// TwinCAT 3 PLC project MotionTemplate
// ProgramVersion: 3.1.4024.0
// libraries:
//   Tc2_MC2, * (Beckhoff Automation GmbH)
//   Tc2_Standard, * (Beckhoff Automation GmbH)
//   Tc2_System, * (Beckhoff Automation GmbH)
//   Tc3_Module, * (Beckhoff Automation GmbH)
// project tree:
//   / PlcTask.TcTTO
//   POUs/ FB_AxisBase.TcPOU, FB_SafetyBase.TcPOU, MAIN.TcPOU
// real-time tasks:
//   TASK PlcTask: cycle T#10ms, priority 20, ADS port 350
// motion (NC):
//   TASK NC-Task 1 SAF: cycle T#2ms, priority 4, ADS port 501
//   TASK NC-Task 1 SVB: cycle T#10ms, priority 8, ADS port 511
//   AXIS Axis 1 (id 1)
//     OtherSettings: AllowMotionCmdToSlave=true
//     encoder EncType=19
//       EncPara: MaxCount=#xffffffff
//     drive DrvType=16
//       DrvPara: MaxCount=#xffffffff, DriveControlDWord=#x00020100
//         Analog: TorqueSetpointScale=10
//         TimeComp: TaskDelayCycles=1
//     controller CtrType=1
//       CtrPara: PriorControlFactor=1
//         Observer: BandWidth=20
//   AXIS AX5_ChA (id 2)
//     Dynamic: Acceleration=8102, Deceleration=8102, Jerk=24306
//     Velo: RefSearch=54, RefSync=54, SlowManual=270, FastManual=1620, Fast=5401, Maximum=5401
//     OtherSettings: AllowMotionCmdToSlave=true
//     encoder EncType=8
//       EncPara: ScaleFactorNumerator=60, ScaleFactorDenominator=1048576, MaxCount=#xffffffff
//     drive DrvType=9
//       DrvPara: MaxCount=#xffffffff, DriveControlDWord=#x00030100
//         Analog: VeloReferenz=5941, TorqueSetpointScale=10
//         TimeComp: TaskDelayCycles=1
//     controller CtrType=1
//       CtrPara: PriorControlFactor=1
//         Observer: BandWidth=20
//   AXIS Axis 3 (id 3)
//     OtherSettings: AllowMotionCmdToSlave=true
//     encoder EncType=8
//       EncPara: MaxCount=#xffffffff
//     drive DrvType=9
//       DrvPara: MaxCount=#xffffffff, DriveControlDWord=#x00030100
//         Analog: TorqueSetpointScale=10
//         TimeComp: TaskDelayCycles=1
//     controller CtrType=1
//       CtrPara: PriorControlFactor=1
//         Observer: BandWidth=20
//   AXIS AX8_ChA (id 4)
//     OtherSettings: AllowMotionCmdToSlave=true
//     encoder EncType=19
//       EncPara: MaxCount=#xffffffff
//     drive DrvType=16
//       DrvPara: MaxCount=#xffffffff, DriveControlDWord=#x00020100
//         Analog: TorqueSetpointScale=10
//         TimeComp: TaskDelayCycles=1
//     controller CtrType=1
//       CtrPara: PriorControlFactor=1
//         Observer: BandWidth=20
// I/O:
//   DEVICE Device 1 (EtherCAT), AmsNetId 5.80.201.232.2.1
//     Term 1 (EK1200) [EK1200-5000 EtherCAT Power supply (2A E-Bus)]
//       Term 2 (ELM7231-9018) [ELM7231-9018 1Ch. Servo Terminal (48 V, 16 A RMS, OCT, STO, Safe Motion, TwinSAFE Logic)]
//         modules: Module 1 (SAFETY)
//       Term 3 (EL4122) [EL4122 2Ch. Ana. Output  4-20mA, 16bit]
//       Term 4 (EL1918) [EL1918, 8Ch. Safety Input 24V, TwinSAFE]
//         modules: Module 1 (FSOE), Module 2 (FSLOGIC)
//       Term 5 (EK1110) [EK1110 EtherCAT extension]
//     Term 6 (EK1100) [EK1100 EtherCAT Coupler (2A E-Bus)]
//       Term 7 (EL6910) [EL6910, TwinSAFE PLC]
//       Term 8 (EL1904) [EL1904, 4 Ch. Safety Input 24V, TwinSAFE]
//         modules: Module 1 (FSOES)
//       Term 11 (EL9011) [EL9011 End Terminal]
//     Drive 9 (AX5206-0000-0214) [AX5206-0000-0214 EtherCAT Drive (SoE, 2 Ch.)]
//       Term 10 (AX5805) [AX5805 (Safety Drive Option)]
//         modules: Module 1 (Safety Process Data, 2 axis), Module 2 (Standard Process Data, 2 axis)
//     Term 22 (AX8620-0000-0102) [AX8620-0000-0102]
//       Drive 23 (AX8206-0210-0107) [AX8206-0210-0107 (2Ch. 6A servo axis, safe-motion, multi-FB)]
//         modules: Device, Device, Device, Device, Device, Device, Device, Device, Device, Device, Device (Safety), Device, Device, Device, Device, Device, Device, Device, Device, Device, Device, Device, Device, Device, Device, Device, Device, Device, Device, Device, Device, Ch A, Ch A, Ch A, Ch A, Ch A, Ch A, Ch A, Ch A, Ch A, Ch A, Ch A, Ch A, Ch A, Ch A, Ch A, Ch A, Ch A, Ch A, Ch A, Ch A, Ch A, Ch A, Ch A, Ch A, Ch A, Ch A, Ch B, Ch B, Ch B, Ch B, Ch B, Ch B, Ch B, Ch B, Ch B, Ch B, Ch B, Ch B, Ch B, Ch B, Ch B, Ch B, Ch B, Ch B, Ch B, Ch B, Ch B, Ch B, Ch B, Ch B, Ch B, Ch B
//         startup 12992:1 := 414D383032312D78427830 // Ch A Motor parameters / Configured motor type
//         startup 24768:0 := FEFF // Ch A Interpolation sub mode select
//         startup 13000:5 := 0200 // Ch A Motor thermal model / Reaction
//         startup 13000:6 := 0000C841 // Ch A Motor thermal model / Partial fraction factor
//         startup 12992:12 := 0000FA45 // Ch A Motor parameters / Motor rated speed
//         startup 12992:13 := C9E5FF3E // Ch A Motor parameters / Motor rated torque
//         startup 24694:0 := F4010000 // Ch A Motor standstill torque
//         startup 24800:0 := D007 // Ch A Positive torque/force limit value
//         startup 24801:0 := D007 // Ch A Negative torque/force limit value
//         startup 12288:6 := 4158383230362D303231302D30303030 // Ch A AxisMain parameters / Configured drive type
//         startup 12867:1 := 9A99593F // Ch A TorqueCtrl parameters / Configured channel rated current
//         startup 12867:2 := 33332340 // Ch A TorqueCtrl parameters / Configured channel peak current
//         startup 12867:7 := 77BE1F40 // Ch A TorqueCtrl parameters / Iuvw max sum
//         startup 24672:0 := 08 // Ch A Modes of operation
//         startup 13023:0 := 0000 // Ch A Motor control mode
//         startup 12864:1 := 0D4D7043 // Ch A TorqueCtrl parameters mappable / Torque control proportional gain q
//         startup 12864:2 := 8A0E7C39 // Ch A TorqueCtrl parameters mappable / Torque control integral action time q
//         startup 12608:1 := FBD1CD3B // Ch A VeloCtrl parameters mappable / Velocity control proportional gain
//         startup 12608:2 := 6F12033C // Ch A VeloCtrl parameters mappable / Velocity control integral action time
//         startup 12608:3 := 00980546 // Ch A VeloCtrl parameters mappable / Bipolar velocity limit value
//         startup 12992:15 := 0100 // Ch A Motor parameters / Motor temperature sensor connection
//         startup 12611:4 := 0400 // Ch A VeloCtrl observer / Observer type
//         startup 24672:0 := 08 // Ch A Modes of operation
//         startup 12296:2 := 00 // Ch A AxisMain parameters encoder direction / Primary encoder direction
//         startup 14016:1 := 414D383131312D78467830 // Ch B Motor parameters / Configured motor type
//         startup 26816:0 := FEFF // Ch B Interpolation sub mode select
//         startup 14024:5 := 0200 // Ch B Motor thermal model / Reaction
//         startup 14024:6 := 0000C841 // Ch B Motor thermal model / Partial fraction factor
//         startup 14016:12 := 00007A45 // Ch B Motor parameters / Motor rated speed
//         startup 14016:13 := CDCE423E // Ch B Motor parameters / Motor rated torque
//         startup 26742:0 := C8000000 // Ch B Motor standstill torque
//         startup 26848:0 := D007 // Ch B Positive torque/force limit value
//         startup 26849:0 := D007 // Ch B Negative torque/force limit value
//         startup 13312:6 := 4158383230362D303231302D30303030 // Ch B AxisMain parameters / Configured drive type
//         startup 13891:1 := 66663640 // Ch B TorqueCtrl parameters / Configured channel rated current
//         startup 13891:2 := CDCC0841 // Ch B TorqueCtrl parameters / Configured channel peak current
//         startup 13891:7 := 77BE1F40 // Ch B TorqueCtrl parameters / Iuvw max sum
//         startup 26720:0 := 08 // Ch B Modes of operation
//         startup 14047:0 := 0000 // Ch B Motor control mode
//         startup 13888:1 := EB27AC40 // Ch B TorqueCtrl parameters mappable / Torque control proportional gain q
//         startup 13888:2 := 8A0E7C39 // Ch B TorqueCtrl parameters mappable / Torque control integral action time q
//         startup 13632:1 := 5DA1B43A // Ch B VeloCtrl parameters mappable / Velocity control proportional gain
//         startup 13632:2 := 6F12033C // Ch B VeloCtrl parameters mappable / Velocity control integral action time
//         startup 13632:3 := 00980546 // Ch B VeloCtrl parameters mappable / Bipolar velocity limit value
//         startup 13635:4 := 0400 // Ch B VeloCtrl observer / Observer type
//         startup 26720:0 := 08 // Ch B Modes of operation
//         startup 13320:2 := 00 // Ch B AxisMain parameters encoder direction / Primary encoder direction
// variable links:
//   Device 1 (EtherCAT) <-> Device 1 (EtherCAT)/Drive 9 (AX5206-0000-0214)/Term 10 (AX5805)
//     Term 6 (EK1100)/Term 7 (EL6910)/ConnectionOutputs/Message_3 RxPDO <-> Module 1 (Safety Process Data, 2 axis)/Inputs (Statusword)/FSOE
//   Device 1 (EtherCAT) <-> Device 1 (EtherCAT)/Term 22 (AX8620-0000-0102)/Drive 23 (AX8206-0210-0107)
//     Term 22 (AX8620-0000-0102)/PSM Controlword for axis/Controlword for axis <-> Device/DeviceMain Outputs/Power supply controlword
//   Device 1 (EtherCAT) <-> Device 1 (EtherCAT)/Term 6 (EK1100)/Term 7 (EL6910)
//     Drive 9 (AX5206-0000-0214)/Term 10 (AX5805)/Module 1 (Safety Process Data, 2 axis)/Outputs (Controlword)/FSOE <-> ConnectionInputs/Message_3 TxPDO
//     Term 6 (EK1100)/Term 8 (EL1904)/Module 1 (FSOES)/RxPDO/FSOE <-> ConnectionInputs/Message_4 TxPDO
//     Term 6 (EK1100)/Term 8 (EL1904)/Module 1 (FSOES)/TxPDO/FSOE <-> ConnectionOutputs/Message_4 RxPDO
//   NC-Task 1 SAF/Axes/AX5_ChA <-> Device 1 (EtherCAT)/Drive 9 (AX5206-0000-0214)
//     Drive/Inputs/In/nDataIn1 <-> AT 1/Following distance
//     Drive/Inputs/In/nDcOutputTime <-> InfoData/DcOutputShift
//     Drive/Inputs/In/nState1 <-> AT 1/Drive status word @bit 8
//     Drive/Inputs/In/nState2 <-> AT 1/Drive status word
//     Drive/Inputs/In/nState4 @bit 1 <-> WcState/InputToggle
//     Drive/Inputs/In/nState4 <-> WcState/WcState
//     Drive/Outputs/Out/nCtrl1 <-> MDT 1/Master control word @bit 8
//     Drive/Outputs/Out/nDataOut1 <-> MDT 1/Position command value
//     Enc/Inputs/In/nDataIn1 <-> AT 1/Position feedback 1 value
//     Enc/Inputs/In/nDcInputTime <-> InfoData/DcInputShift
//     Enc/Inputs/In/nState4 @bit 1 <-> WcState/InputToggle
//     Enc/Inputs/In/nState4 <-> WcState/WcState
//   NC-Task 1 SAF/Axes/AX8_ChA <-> Device 1 (EtherCAT)/Term 22 (AX8620-0000-0102)/Drive 23 (AX8206-0210-0107)
//     Drive/Inputs/In/nDataIn1 <-> Ch A/Ch A PositionControl Inputs/Ch A Following error actual value
//     Drive/Inputs/In/nDcOutputTime <-> InfoData/DcOutputShift
//     Drive/Inputs/In/nState1 <-> Ch A/Ch A AxisMain Inputs/Ch A Statusword
//     Drive/Inputs/In/nState2 <-> Ch A/Ch A AxisMain Inputs/Ch A Statusword @bit 8
//     Drive/Inputs/In/nState4 @bit 1 <-> WcState/InputToggle0
//     Drive/Inputs/In/nState4 <-> WcState/WcState0
//     Drive/Outputs/Out/nCtrl1 <-> Ch A/Ch A AxisMain Outputs/Ch A Controlword
//     Drive/Outputs/Out/nCtrl2 <-> Ch A/Ch A AxisMain Outputs/Ch A Controlword @bit 8
//     Drive/Outputs/Out/nDataOut1 <-> Ch A/Ch A Interpolator Outputs/Ch A Target position
//     Drive/Outputs/Out/nDataOut2 <-> Ch A/Ch A Interpolator Outputs/Ch A Target velocity
//     Enc/Inputs/In/nDataIn1 <-> Ch A/Ch A AxisMain Inputs/Ch A Position actual value
//     Enc/Inputs/In/nDcInputTime <-> InfoData/DcInputShift
//     Enc/Inputs/In/nState2 @bit 5 <-> Ch A/Ch A AxisMain Inputs/Position actual value invalid
//     Enc/Inputs/In/nState4 @bit 1 <-> WcState/InputToggle0
//     Enc/Inputs/In/nState4 <-> WcState/WcState0
//   NC-Task 1 SAF/Axes/Axis 1 <-> Device 1 (EtherCAT)/Term 1 (EK1200)/Term 2 (ELM7231-9018)
//     Drive/Inputs/In/nDataIn1 <-> DRV Following error actual value/Following error actual value
//     Drive/Inputs/In/nDcOutputTime <-> InfoData/DcOutputShift
//     Drive/Inputs/In/nState1 <-> DRV Statusword/Statusword
//     Drive/Inputs/In/nState2 <-> DRV Statusword/Statusword @bit 8
//     Drive/Inputs/In/nState4 @bit 1 <-> WcState/InputToggle0
//     Drive/Inputs/In/nState4 <-> WcState/WcState0
//     Drive/Outputs/Out/nCtrl1 <-> DRV Controlword/Controlword
//     Drive/Outputs/Out/nCtrl2 <-> DRV Controlword/Controlword @bit 8
//     Drive/Outputs/Out/nDataOut1 <-> DRV Target position/Target position
//     Enc/Inputs/In/nDataIn1 <-> FB Position/Position
//     Enc/Inputs/In/nDcInputTime <-> InfoData/DcInputShift
//     Enc/Inputs/In/nState4 @bit 1 <-> WcState/InputToggle0
//     Enc/Inputs/In/nState4 <-> WcState/WcState0
//   NC-Task 1 SAF/Axes/Axis 3 <-> Device 1 (EtherCAT)/Drive 9 (AX5206-0000-0214)
//     Drive/Inputs/In/nDataIn1 <-> AT 2/Following distance
//     Drive/Inputs/In/nDcOutputTime <-> InfoData/DcOutputShift
//     Drive/Inputs/In/nState1 <-> AT 2/Drive status word @bit 8
//     Drive/Inputs/In/nState2 <-> AT 2/Drive status word
//     Drive/Inputs/In/nState4 @bit 1 <-> WcState/InputToggle
//     Drive/Inputs/In/nState4 <-> WcState/WcState
//     Drive/Outputs/Out/nCtrl1 <-> MDT 2/Master control word @bit 8
//     Drive/Outputs/Out/nDataOut1 <-> MDT 2/Position command value
//     Enc/Inputs/In/nDataIn1 <-> AT 2/Position feedback 1 value
//     Enc/Inputs/In/nDcInputTime <-> InfoData/DcInputShift
//     Enc/Inputs/In/nState4 @bit 1 <-> WcState/InputToggle
//     Enc/Inputs/In/nState4 <-> WcState/WcState
//   MotionTemplate/MotionTemplate Instance <-> Device 1 (EtherCAT)/Term 6 (EK1100)/Term 7 (EL6910)
//     PlcTask Outputs/MAIN.safety.b_errAck_a <-> StandardOutputs/Standard In Var 1
//     PlcTask Outputs/MAIN.safety.b_errAck_b <-> StandardOutputs/Standard In Var 5
//     PlcTask Outputs/MAIN.safety.b_run_a <-> StandardOutputs/Standard In Var 2

CONFIGURATION MotionTemplate
    RESOURCE PLC ON TwinCAT3
        TASK PlcTask(INTERVAL := T#10ms, PRIORITY := 20);
        PROGRAM MAIN WITH PlcTask : MAIN;
    END_RESOURCE
END_CONFIGURATION

// ---- POUs/MAIN.TcPOU
PROGRAM MAIN
VAR
	safety	: FB_SafetyBase;	

	ax5_chA : FB_AxisBase;
	//ax8_chA : FB_AxisBase;
END_VAR

safety();
ax5_chA();
//ax8_chA();

END_PROGRAM

// ---- POUs/FB_SafetyBase.TcPOU
FUNCTION_BLOCK FB_SafetyBase
VAR_INPUT
	b_start : BOOL;
	t_delay : TIME := T#500MS;
END_VAR
VAR_OUTPUT
END_VAR
VAR
	b_run_a AT %Q* : BOOL := TRUE;
	b_run_b AT %Q* : BOOL := TRUE;
	b_run_c AT %Q* : BOOL := TRUE;
	b_run_d AT %Q* : BOOL := TRUE;
	
	b_errAck_a AT %Q* : BOOL;
	b_errAck_b AT %Q* : BOOL;
	b_errAck_c AT %Q* : BOOL;
	b_errAck_d AT %Q* : BOOL;
	
	m_r_trig 		: R_TRIG;
	m_n_state 		: UINT;
	m_n_next_state	: UINT;
	m_n_ton 	: TON;
END_VAR

m_r_trig(CLK:= b_start, Q=> );

IF m_r_trig.Q THEN
	m_n_state := 10;
END_IF

CASE m_n_state OF
	0: // Idle
		b_start := FALSE;
		
	10:
		b_errAck_a := TRUE;
		m_n_state := 90;
		m_n_next_state := 11;
		
	11:
		b_errAck_a 		:= FALSE;
		m_n_state 		:= 90;
		m_n_next_state 	:= 20;
		
	20:
		b_errAck_b := TRUE;
		m_n_state := 90;
		m_n_next_state := 21;
		
	21:
		b_errAck_b 		:= FALSE;
		m_n_state 		:= 90;
		m_n_next_state 	:= 30;
		
	30:
		b_errAck_c := TRUE;
		m_n_state := 90;
		m_n_next_state := 31;
		
	31:
		b_errAck_c 		:= FALSE;
		m_n_state 		:= 90;
		m_n_next_state 	:= 40;

	40:
		b_errAck_d := TRUE;
		m_n_state := 90;
		m_n_next_state := 41;
		
	41:
		b_errAck_d 		:= FALSE;
		m_n_state 		:= 90;
		m_n_next_state 	:= 0;	
		
	90:
		m_n_ton(IN:= TRUE, PT:= t_delay);
		IF m_n_ton.Q THEN
			m_n_ton(IN:= FALSE);
			m_n_state := m_n_next_state;
		END_IF
END_CASE

END_FUNCTION_BLOCK

// ---- POUs/FB_AxisBase.TcPOU
FUNCTION_BLOCK FB_AxisBase
VAR_INPUT
	bPowerEnable 	: BOOL := TRUE;
	bPosEnable		: BOOL := TRUE;
	bNegEnable		: BOOL := TRUE;
	bStop			: BOOL;
	bReset 			: BOOL;
	fOverride		: LREAL := 100.0;
END_VAR
VAR_OUTPUT
	bAxisRdy		: BOOL;
	bError			: BOOL;
	nErrId			: UDINT;
END_VAR
VAR
	m_axis		: AXIS_REF;	

	m_fb_power 	: MC_Power;
	m_fb_reset	: MC_Reset;
	m_fb_stop  	: MC_Stop;
	m_fb_state	: MC_ReadStatus;

	m_axis_status 	: ST_AxisStatus;
	m_state			: ST_McOutputs;
	st_fbMcStopOut	: ST_McOutputs;
	
END_VAR

m_fb_state(Axis:= m_axis, Enable:= TRUE);


m_fb_power(
	Axis 				:= m_axis,
	Enable 				:= bPowerEnable,
	Override 			:= fOverride,
	Enable_Positive 	:= bPosEnable,
	Enable_Negative 	:= bNegEnable,
);
	
m_fb_reset(
	Axis := m_axis,
	Execute := bReset
	);

	
m_fb_stop(
	Axis := m_axis,
	Execute := bStop,
	);


bStop 	:= FALSE;
bReset 	:= FALSE;

bAxisRdy	:= m_fb_power.Status;
bError 		:= m_fb_power.Error 		OR m_fb_reset.Error		OR m_fb_stop.Error OR m_fb_state.Error;
nErrId 		:= m_fb_power.ErrorID OR m_fb_reset.ErrorID	OR m_fb_stop.ErrorID OR m_fb_state.ErrorID;

END_FUNCTION_BLOCK
